(* PLC project Blank Project, Blank Blank 1.0 *)
(* stored: creationDateTime 2016-05-18T21:14:07, modificationDateTime 2017-02-10T21:03:05 *)

FUNCTION_BLOCK BlockTest
  VAR_INPUT
    In : BOOL;
  END_VAR
  VAR_OUTPUT
    Out : BOOL;
  END_VAR
  VAR
    MYARRAY : ARRAY[0..5] OF INT;
  END_VAR

            In := Out;

MYARRAY[0] := 1;
MYARRAY[1] := 2;
MYARRAY[2] := 3;
MYARRAY[3] := 4;
MYARRAY[4] := 5;
MYARRAY[5] := 7;
          
END_FUNCTION_BLOCK

PROGRAM My_Program
  VAR
    iniciar : BOOL := FALSE;
    parar : BOOL := FALSE;
    lamp : BOOL;
    test1 : SINT := 15;
    test2 : INT := 15;
    test3 : DINT := 15;
    test4 : LINT := 15;
    test5 : USINT := 15;
    test6 : UINT := 15;
    test7 : UDINT := 15;
    test8 : ULINT := 15;
    test9 : REAL := 15.0;
    test10 : LREAL := 15.0;
    test11 : TIME := T#14.7s;
    test12 : TIME := TIME#14ms;
    test13 : TIME := t#5d_14h_12m_18s_3.5ms;
    test14 : DATE := D#1984-06-25;
    test15 : TOD := TOD#15:36:55.36;
    test16 : DT := DT#1984-06-25-15:36:55.36;
    test17 : STRING := 'HELLO';
    test18 : BYTE := 15;
    test19 : WORD := 15;
    test20 : DWORD := 15;
    test21 : LWORD := 12315555;
    BlockTest0 : BlockTest;
    InputTest : BOOL := TRUE;
    OutputTest : BOOL;
    TestARRAY : ARRAY[0..4] OF SINT := [1, 2, 3, 4, 5];
    TestARRAY0 : ARRAY[0..4] OF SINT := [5(4)];
  END_VAR

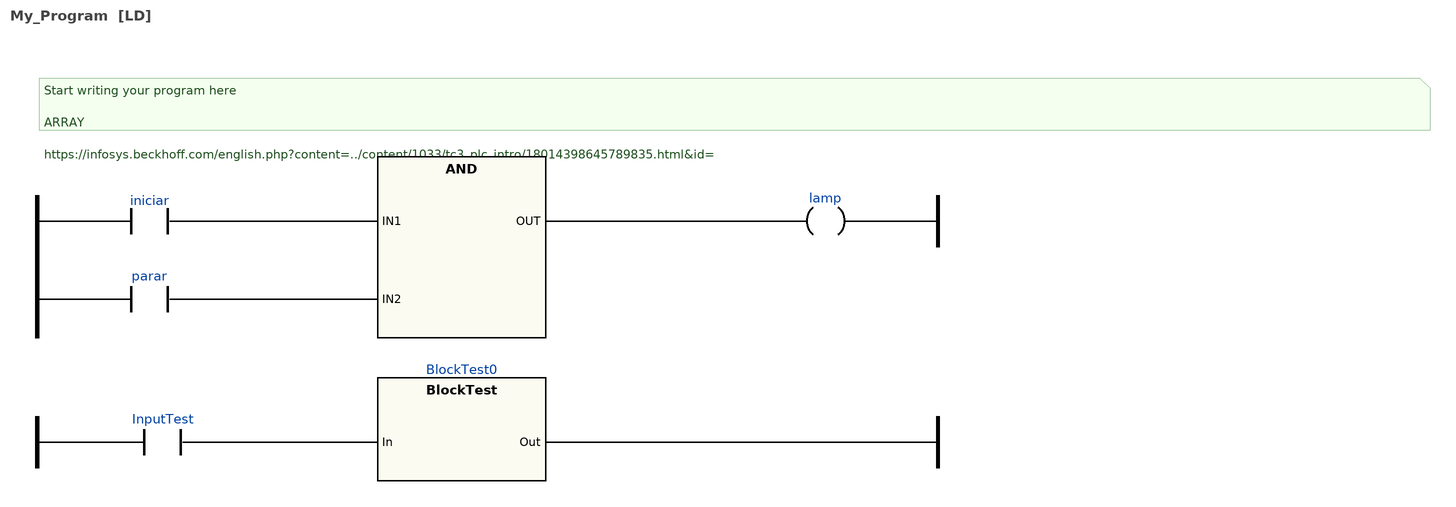
(* LD diagram, written out as Structured Text *)
(* Start writing your program here

ARRAY

https://infosys.beckhoff.com/english.php?content=../content/1033/tc3_plc_intro/18014398645789835.html&id= *)
lamp := iniciar AND parar;
BlockTest0(In := InputTest);
END_PROGRAM

CONFIGURATION STD_CONF
  RESOURCE STD_RESSOURCE ON PLC
    TASK TaskMain(INTERVAL := T#50ms, PRIORITY := 0);
    PROGRAM Inst0 WITH TaskMain : My_Program;
  END_RESOURCE
END_CONFIGURATION
